PROGRAM OperatingModes
VAR
	AuxStopping:Modes;
END_VAR

CASE GVL.Mode OF
	
	// Emergency stop
	Modes.STOP_EM:
		IF HMI.Bt_Rearm THEN
			gvl.Mode := modes.STOP_OP;
		END_IF
	
	// Operative stop
	Modes.STOP_OP:
		IF HMI.Bt_EmStop THEN
			GVL.Mode := Modes.STOP_EM;
		END_IF
		IF HMI.Bt_Run AND HMI.S_ManAuto THEN
			GVL.Mode := Modes.AUTO;
			GVL.State:=0;
		END_IF
		IF NOT HMI.S_ManAuto THEN
			GVL.Mode := Modes.MAN;
		END_IF
		
	// Automatic
	Modes.AUTO:
		IF HMI.Bt_EmStop THEN
			GVL.Mode := Modes.STOP_EM;
		END_IF
		IF NOT HMI.S_ManAuto THEN
			GVL.Mode := Modes.MAN;
		END_IF
		IF HMI.Bt_Stop THEN
			GVL.Mode := Modes.Stopping;
			AuxStopping := Modes.STOP_OP;
		END_IF
		
	// Manual
	Modes.MAN:
		IF HMI.Bt_EmStop THEN
			GVL.Mode := Modes.STOP_EM;
		END_IF
		IF HMi.S_ManAuto THEN
			GVL.Mode := Modes.STOP_OP;
		END_IF	
		
	// Stopping
	Modes.Stopping:
		MC.Exec_Stop:= TRUE;
		IF (Motion.FB_Stop.Done AND Motion.FB_StopPuller.Done AND Motion.FB_StopPullerVirtual.Done AND Motion.FB_GearOut.Done) OR MC.Extruder.Status.Error OR MC.Puller.Status.Error OR MC.PullerVirtual.Status.Error THEN
			GVL.Mode := AuxStopping;
		END_IF
END_CASE

// Axis Power when not in stop
IF GVL.Mode = Modes.AUTO OR GVL.Mode = Modes.Stopping THEN
	MC.En_Power := TRUE;
END_IF

END_PROGRAM

(* stored: Version 1.1.0.1, ProductVersion 3.1.4024.9
   POU OperatingModes: Id {041e3654-c2e6-485e-9be9-b8cb759cbbc6}, SpecialFunc None *)
